// SIMATIC S7-200 SMART project (STEP 7-Micro/WIN SMART), CPU SR40

SYMBOL_TABLE 系统符号
Always_On        SM0.0    // 始终接通
First_Scan_On    SM0.1    // 仅在第一个扫描周期时接通
END_SYMBOL_TABLE

ORGANIZATION_BLOCK MAIN:OB1
TITLE=程序注释
BEGIN
Network 1
// 程序段注释
LD     First_Scan_On:SM0.1   //首次扫描时
MOVW   16#E00, MW0           //设置彩灯初始值，Q0.1～Q0.3对应的灯亮
Network 2
LDN    T37
TON    T37, +20              //产生周期为2s的移位脉冲
?000
Network 3
LD     T37                   //移位时间到
LPS
RLW    MW0, 1                //彩灯左移1位
A      M1.2                  //将M1.1移入M1.2的数据传送到M0.0
S      M0.0, 1
LPP
AN     M1.2
R      M0.0, 1
Network 4
LD     Always_On:SM0.0
MOVB   MB0, QB0
Network 5
LD     M1.1
=      Q1.1
Network 6
LD     M1.0
=      Q1.0
END_ORGANIZATION_BLOCK
